% RSLogix 500 project P7_BAK048.RSS, saved by version 12.00.00.00 %
PROJECT "UNTITLED"    % processor: Bul.1763 MicroLogix 1100 Series B %

PROGRAM FILES
  LAD 2 "MAIN"  3 rungs
  LAD 3 "DIGITAL IO"  3 rungs
  LAD 4 "CONTROLS"  14 rungs

DATA FILES
  O0 OUTPUT  4 elements
  I1 INPUT  6 elements
  S2 STATUS  66 elements
  B3 BINARY  1 elements
  T4 TIMER  4 elements
  C5 COUNTER  2 elements
  R6 CONTROL  1 elements
  N7 INTEGER  13 elements
  F8 FLOAT  5 elements

LADDER 2 "MAIN"
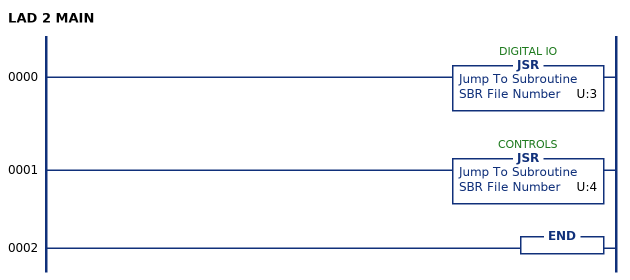
% Rung: 0 %
SOR JSR U:3 EOR
%   U:3  "DIGITAL IO" %
% Rung: 1 %
SOR JSR U:4 EOR
%   U:4  "CONTROLS" %
% Rung: 2 %
SOR END EOR

LADDER 3 "DIGITAL IO"
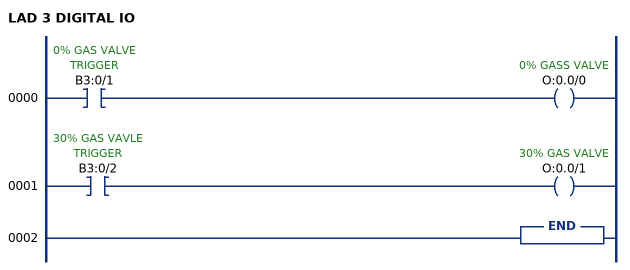
% Rung: 0 %
SOR XIC B3:0/1 OTE O:0.0/0 EOR
%   B3:0/1  "0% GAS VALVE TRIGGER" %
%   O:0.0/0  "0% GASS VALVE" %
% Rung: 1 %
SOR XIC B3:0/2 OTE O:0.0/1 EOR
%   B3:0/2  "30% GAS VAVLE TRIGGER" %
%   O:0.0/1  "30% GAS VALVE" %
% Rung: 2 %
SOR END EOR

LADDER 4 "CONTROLS"
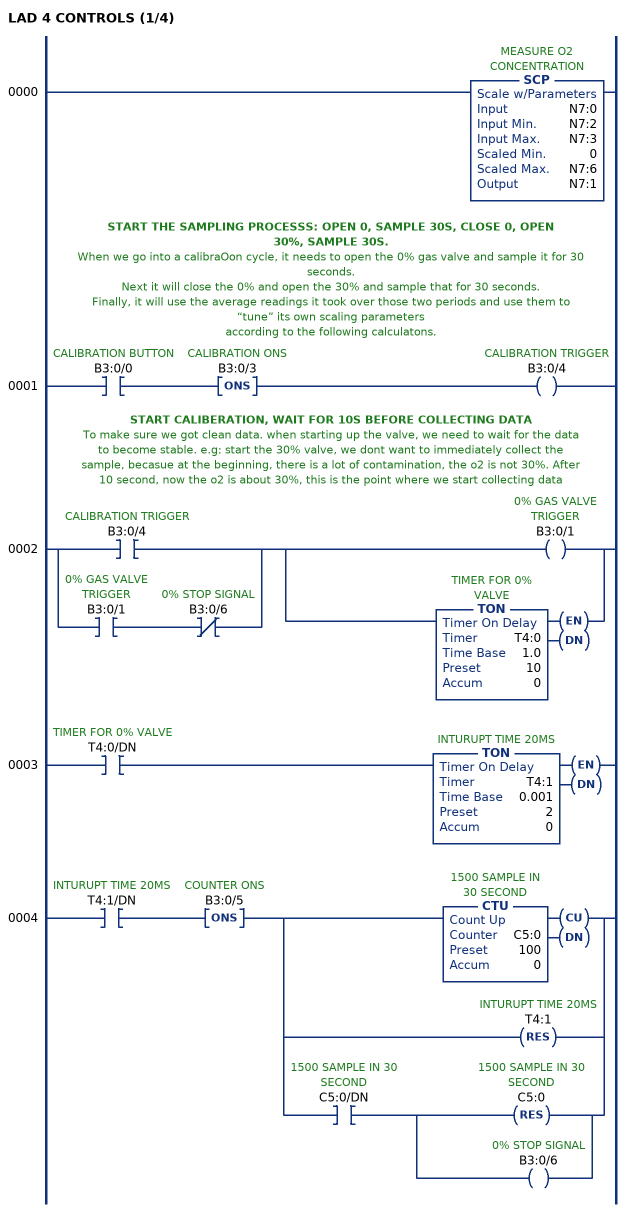
% Rung: 0 %
SOR SCP N7:0 N7:2 N7:3 0 N7:6 N7:1 EOR
%   N7:0  "O2 SENSOR INPUT SIGNAL" %
%   N7:2  "O2 INPUT MIN" %
%   N7:3  "O2 INPUT MAX" %
%   N7:6  "(N-1)*A[N-1]" %
%   N7:1  "MEASURE O2 CONCENTRATION" %
% Rung: 1 %
% TITLE: START THE SAMPLING PROCESSS: OPEN 0, SAMPLE 30S, CLOSE 0, OPEN 30%, SAMPLE 30S. %
% When we go into a calibraOon cycle, it needs to open the 0% gas valve and sample it for 30 seconds.
% Next it will close the 0% and open the 30% and sample that for 30 seconds.
% Finally, it will use the average readings it took over those two periods and use them to “tune” its own scaling parameters
% according to the following calculatons. %
SOR XIC B3:0/0 ONS B3:0/3 OTE B3:0/4 EOR
%   B3:0/0  "CALIBRATION BUTTON" %
%   B3:0/3  "CALIBRATION ONS" %
%   B3:0/4  "CALIBRATION TRIGGER" %
% Rung: 2 %
% TITLE: START CALIBERATION, WAIT FOR 10S BEFORE COLLECTING DATA %
% To make sure we got clean data. when starting up the valve, we need to wait for the data to become stable. e.g: start the 30% valve, we dont want to immediately collect the sample, becasue at the beginning, there is a lot of contamination, the o2 is not 30%. After 10 second, now the o2 is about 30%, this is the point where we start collecting data %
SOR BST XIC B3:0/4 NXB XIC B3:0/1 XIO B3:0/6 BND BST OTE B3:0/1 NXB TON T4:0 1.0 10 0 BND EOR
%   B3:0/4  "CALIBRATION TRIGGER" %
%   B3:0/1  "0% GAS VALVE TRIGGER" %
%   B3:0/6  "0% STOP SIGNAL" %
%   T4:0  "TIMER FOR 0% VALVE" %
% Rung: 3 %
SOR XIC T4:0/DN TON T4:1 0.001 2 0 EOR
%   T4:0  "TIMER FOR 0% VALVE" %
%   T4:1  "INTURUPT TIME 20MS" %
% Rung: 4 %
SOR XIC T4:1/DN ONS B3:0/5 BST CTU C5:0 100 0 NXB RES T4:1 NXB XIC C5:0/DN BST RES C5:0 NXB OTE B3:0/6 BND BND EOR
%   T4:1  "INTURUPT TIME 20MS" %
%   B3:0/5  "COUNTER ONS" %
%   C5:0  "1500 SAMPLE IN 30 SECOND" %
%   B3:0/6  "0% STOP SIGNAL" %

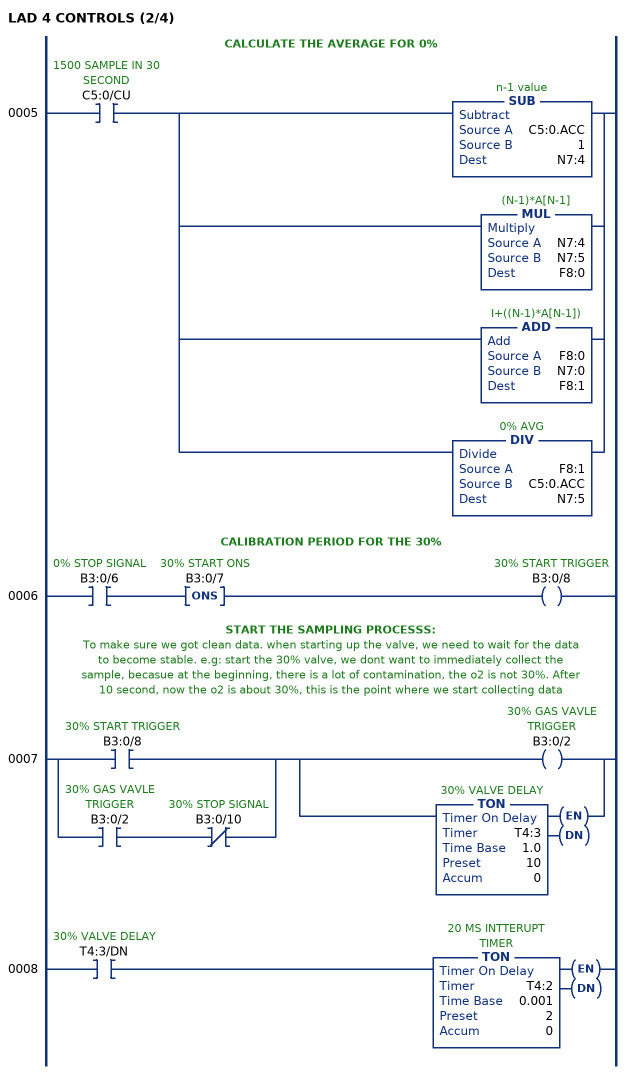
% Rung: 5 %
% TITLE: CALCULATE THE AVERAGE FOR 0% %
SOR XIC C5:0/CU BST SUB C5:0.ACC 1 N7:4 NXB MUL N7:4 N7:5 F8:0 NXB ADD F8:0 N7:0 F8:1 NXB DIV F8:1 C5:0.ACC N7:5 BND EOR
%   C5:0  "1500 SAMPLE IN 30 SECOND" %
%   N7:4  "n-1 value" %
%   N7:5  "0% AVG" %
%   F8:0  "(N-1)*A[N-1]" %
%   N7:0  "O2 SENSOR INPUT SIGNAL" %
%   F8:1  "I+((N-1)*A[N-1])" %
% Rung: 6 %
% TITLE: CALIBRATION PERIOD FOR THE 30% %
SOR XIC B3:0/6 ONS B3:0/7 OTE B3:0/8 EOR
%   B3:0/6  "0% STOP SIGNAL" %
%   B3:0/7  "30% START ONS" %
%   B3:0/8  "30% START TRIGGER" %
% Rung: 7 %
% TITLE: START THE SAMPLING PROCESSS: %
% To make sure we got clean data. when starting up the valve, we need to wait for the data to become stable. e.g: start the 30% valve, we dont want to immediately collect the sample, becasue at the beginning, there is a lot of contamination, the o2 is not 30%. After 10 second, now the o2 is about 30%, this is the point where we start collecting data %
SOR BST XIC B3:0/8 NXB XIC B3:0/2 XIO B3:0/10 BND BST OTE B3:0/2 NXB TON T4:3 1.0 10 0 BND EOR
%   B3:0/8  "30% START TRIGGER" %
%   B3:0/2  "30% GAS VAVLE TRIGGER" %
%   B3:0/10  "30% STOP SIGNAL" %
%   T4:3  "30% VALVE DELAY" %
% Rung: 8 %
SOR XIC T4:3/DN TON T4:2 0.001 2 0 EOR
%   T4:3  "30% VALVE DELAY" %
%   T4:2  "20 MS INTTERUPT TIMER" %

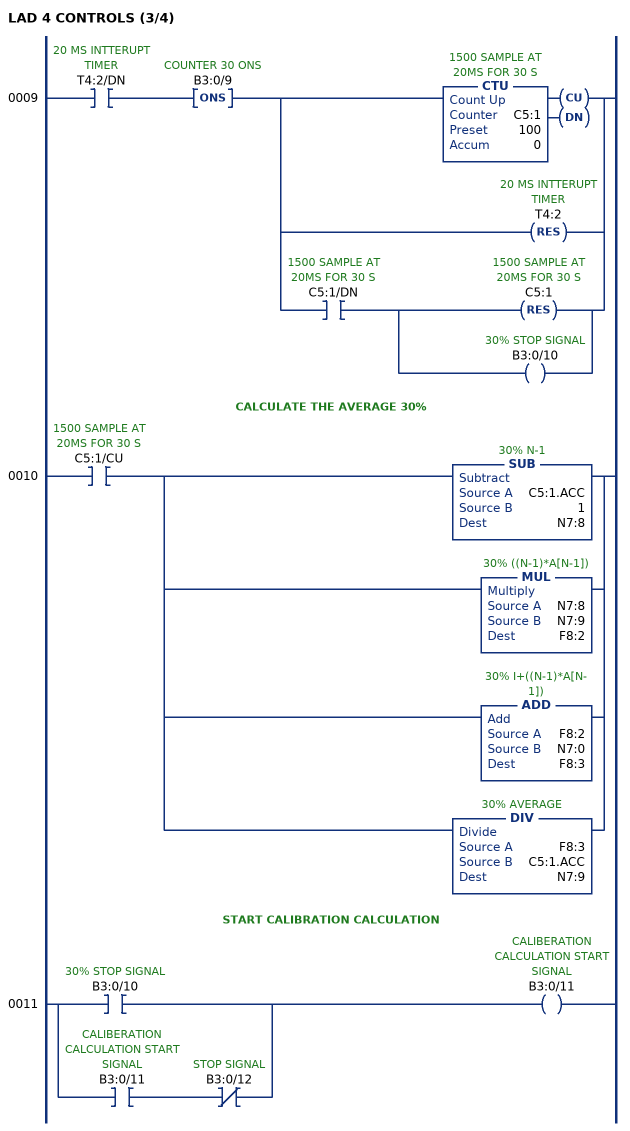
% Rung: 9 %
SOR XIC T4:2/DN ONS B3:0/9 BST CTU C5:1 100 0 NXB RES T4:2 NXB XIC C5:1/DN BST RES C5:1 NXB OTE B3:0/10 BND BND EOR
%   T4:2  "20 MS INTTERUPT TIMER" %
%   B3:0/9  "COUNTER 30 ONS" %
%   C5:1  "1500 SAMPLE AT 20MS FOR 30 S" %
%   B3:0/10  "30% STOP SIGNAL" %
% Rung: 10 %
% TITLE: CALCULATE THE AVERAGE 30% %
SOR XIC C5:1/CU BST SUB C5:1.ACC 1 N7:8 NXB MUL N7:8 N7:9 F8:2 NXB ADD F8:2 N7:0 F8:3 NXB DIV F8:3 C5:1.ACC N7:9 BND EOR
%   C5:1  "1500 SAMPLE AT 20MS FOR 30 S" %
%   N7:8  "30% N-1" %
%   N7:9  "30% AVERAGE" %
%   F8:2  "30% ((N-1)*A[N-1])" %
%   N7:0  "O2 SENSOR INPUT SIGNAL" %
%   F8:3  "30% I+((N-1)*A[N-1])" %
% Rung: 11 %
% TITLE: START CALIBRATION CALCULATION %
SOR BST XIC B3:0/10 NXB XIC B3:0/11 XIO B3:0/12 BND OTE B3:0/11 EOR
%   B3:0/10  "30% STOP SIGNAL" %
%   B3:0/11  "CALIBERATION CALCULATION START SIGNAL" %
%   B3:0/12  "STOP SIGNAL" %

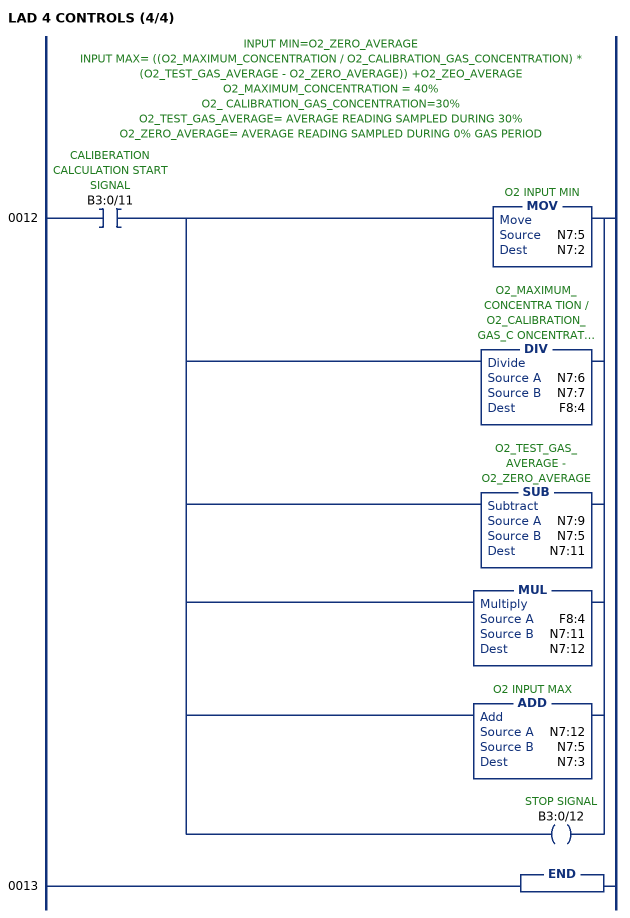
% Rung: 12 %
% INPUT MIN=O2_ZERO_AVERAGE
% INPUT MAX= ((O2_MAXIMUM_CONCENTRATION / O2_CALIBRATION_GAS_CONCENTRATION) * (O2_TEST_GAS_AVERAGE - O2_ZERO_AVERAGE)) +O2_ZEO_AVERAGE
% O2_MAXIMUM_CONCENTRATION = 40%
% O2_ CALIBRATION_GAS_CONCENTRATION=30%
% O2_TEST_GAS_AVERAGE= AVERAGE READING SAMPLED DURING 30%
% O2_ZERO_AVERAGE= AVERAGE READING SAMPLED DURING 0% GAS PERIOD %
SOR XIC B3:0/11 BST MOV N7:5 N7:2 NXB DIV N7:6 N7:7 F8:4 NXB SUB N7:9 N7:5 N7:11 NXB MUL F8:4 N7:11 N7:12 NXB ADD N7:12 N7:5 N7:3 NXB OTE B3:0/12 BND EOR
%   B3:0/11  "CALIBERATION CALCULATION START SIGNAL" %
%   N7:5  "0% AVG" %
%   N7:2  "O2 INPUT MIN" %
%   N7:6  "(N-1)*A[N-1]" %
%   N7:7  "I+((N-1)*A[N-1])" %
%   F8:4  "O2_MAXIMUM_CONCENTRA TION / O2_CALIBRATION_GAS_C ONCENTRATION" %
%   N7:9  "30% AVERAGE" %
%   N7:11  "O2_TEST_GAS_AVERAGE - O2_ZERO_AVERAGE" %
%   N7:3  "O2 INPUT MAX" %
%   B3:0/12  "STOP SIGNAL" %
% Rung: 13 %
SOR END EOR

OTHER DOCUMENTED ADDRESSES
  N7:10  F8  "O2_MAXIMUM_CONCENTRA TION / O2_CALIBRATION_GAS_C ONCENTRATION"

COMMENTS NOT ATTACHED TO A CURRENT RUNG
  N7:2: INPUT MIN=O2_ZERO_AVERAGE
    INPUT MAX= ((O2_MAXIMUM_CONCENTRATION / O2_CALIBRATION_GAS_CONCENTRATION) * (O2_TEST_GAS_AVERAGE - O2_ZERO_AVERAGE)) +O2_ZEO_AVERAGE
    O2_MAXIMUM_CONCENTRATION = 40%
    O2_ CALIBRATION_GAS_CONCENTRATION=30%
    O2_TEST_GAS_AVERAGE= AVERAGE READING SAMPLED DURING 30%
    O2_ZERO_AVERAGE= AVERAGE READING SAMPLED DURING 0% GAS PERIOD

DATA TABLE (non-zero values as saved)
DATA T4
% .PRE .ACC %
% T4:0 % 10 0
% T4:1 % 2 0
% T4:2 % 2 0
% T4:3 % 10 0
DATA C5
% .PRE .ACC %
% C5:0 % 100 0
% C5:1 % 100 0
DATA N7
% N7:0 % 0 0 0 16383 0 0 40 30 0 0
